// TIA Portal V19 export
DATA_BLOCK "Connect_DB"   // DB7
{ S7_Optimized_Access := 'TRUE' }
// stored: MemoryReserve 100
   VAR
      "Out to 1200" : Int;
   END_VAR
BEGIN
END_DATA_BLOCK
